(* CoDeSys 2.3.9.47 project: mqtt.pro *)
(* Libraries: Z:\Users\oedemis\Downloads\WagoLibModbus_IP_01.lib 11.2.16 18:05:40, C:\Program Files\WAGO Software\CoDeSys V2.3\Targets\WAGO\Libraries\32_Bit\oscat_basic_333.lib 9.2.16 18:15:54, WagoLibEthernet_01.lib 11.2.16 18:05:44, SysLibSockets.lib 22.5.14 16:16:32, Standard.lib 20.5.14 08:13:26, Iecsfc.lib 16.5.13 14:00:50, SYSLIBCALLBACK.LIB 16.5.13 14:00:50 *)

(* PLC configuration (modules and I/O channels)
K-Bus [K_Bus] node 0, in %IB0 out %QB0 {KbusBusMode = 1; KbusCycleTime = 10000; KbusThreadPriority = 0; KbusSetOutputsToZeroOnApplicationStop = 1}
Modbus variables [PFC200MODBUS] node 1, in %IB0 out %QB0 {PlcStopBehaviour = 1; FiledbusErrorBehaviour = 1; TcpOperation = 1; TcpPort = 502; TcpTimeout = 600; UdpOperation = 1; UdpPort = 502; RtuOperation = 0; NodeId = 1; ResponseTimeout = 5000; Interface = 0; Baud = 115200; StopBits = 1; Parity = 1; FlowCtrl = 0; PhysInterface = 0}
unused [PFC200CANOPEN_UNUSED] node 2, in %IB6000 out %QB6000
Modbus-Master [MB_MASTER] node 3, in %IB0 out %QB0
*)

(* Task configuration *)
TASK Schedule (PRIORITY := 31, INTERVAL := T#100ms);
	PLC_PRG();
END_TASK

(* Global variable list: Globale_Variablen *)
VAR_GLOBAL
	xxSubscribe: BOOL := TRUE;
	xxPublish : BOOL     := TRUE;
	SubPubState : INT;
END_VAR

(* Data type *)
TYPE Buffer :
STRUCT
	data : ARRAY [0..MAX_RECEIVE_TCP_CLIENT] OF BYTE;
	iPos : DWORD := 0;
END_STRUCT
END_TYPE

(* Data type *)
TYPE ConnectFlags :
STRUCT
	xUsername     : BOOL;
	xPassword     : BOOL;
	xWillRetain   : BOOL;
	xWillQoS1     : BOOL;
    xWillQoS2     : BOOL;
	xWillFlag     : BOOL;
	xCleanSession : BOOL;
END_STRUCT
END_TYPE

(* Data type *)
TYPE FixedHeader :
STRUCT
	bMessageType : BYTE := 16#00;
	xDUP_FLAG    : BOOL := FALSE;
	xQos         : BYTE := 16#00; (*0,1,2*)
	xRetain      : BOOL := FALSE;
END_STRUCT
END_TYPE

(* Data type *)
TYPE FixedHeaderSub :
STRUCT
	bMessageType : BYTE := 8;
	xReserved         : BYTE := 2;
END_STRUCT
END_TYPE

(* Data type *)
TYPE Payload :
STRUCT
	data : ARRAY [0..30] OF BYTE;
	iPos : DWORD := 0;
END_STRUCT
END_TYPE

(* POU PLC_PRG, ST *)
PROGRAM PLC_PRG
VAR
	mqttClient: MQTT_Client;
	xPublish: BOOL;
	xSubscribe: BOOL;

	mqttClientFeedIN : MQTT_Client;
	xPublishFeedIN : BOOL;
	xSubscribeFeedIN : BOOL;

	mqttClient2 : MQTT_Client;
	xPublish2 : BOOL;
	xSubscribe2 : BOOL;

	(*Modbus Communication*)
	KOMMU_E: ETHERNET_MODBUSMASTER_TCP;
	Receive_Data: ARRAY [0..5] OF WORD;
	Transmit_Data: ARRAY [0..3] OF WORD;
	TON1:TON;
	diActivePowerSetpoint:DINT;
	xSend:BOOL := TRUE;

	(*test variables*)
	dummy:DATE_AND_TIME;
	str:STRING;
	x:DATE_AND_TIME;
	y:DATE_AND_TIME;
	z:INT;
END_VAR
mqttClient(
xPublish := xxPublish, (* I/O variable to publish to a TOPIC *)
xSubscribe := xxSubscribe,  (* NOT SUPPORTED, but must be here for I/O *)
sIP:='10.210.10.60', (* IP of the MQTT Broker *)
wPortNumber:=1883,  (* PORT of the MQTT Broker *)
(* AUTH: When no authentication is needed, leave the following fields Blank *)
sUsername:='',  (* Username to connect with the MQTT Broker *)
sPassword:='' (* password to connect with the MQTT Broker *)
);

(*mqttClient.sTopic := 'residual/2015-02-13 09:00:00';*)
mqttClient.sTopic := 'residual/+';
mqttClient.sQoS := 16#00;
mqttClient.pTopic := 'pub';
mqttClient.pQoS := 16#00;
mqttClient.pRetained := FALSE;
mqttClient.pPayload := 'wow';


dummy := STRING_TO_DT('DT#2015-02-13-09:00:15');
str:=DT_TO_STRING(DT#1998-02-13-14:20);
x:= SET_DT(
	year := 2015,
	month := 02,
	day := 13  ,
	HOUR := 09,
	MINUTE := 00,
	SECOND := 00);

y:= SET_DT(
	year := 2015,
	month := 02,
	day := 13  ,
	HOUR := 09,
	MINUTE := 00,
	SECOND := 15);

z := DT_TO_INT(y)-DT_TO_INT(x);

(*z:=SECOND_OF_DT(x) - SECOND_OF_DT(y);*)



(*mqttClientFeedIN(
xPublish := xPublishFeedIN, (* I/O variable to publish to a TOPIC *)
xSubscribe := xPublishFeedIN,  (* NOT SUPPORTED, but must be here for I/O *)
sIP:='10.210.10.60', (* IP of the MQTT Broker *)
wPortNumber:=1883,  (* PORT of the MQTT Broker *)
(* AUTH: When no authentication is needed, leave the following fields Blank *)
sUsername:='',  (* Username to connect with the MQTT Broker *)
sPassword:='' (* password to connect with the MQTT Broker *)
);
mqttClientFeedIN.sTopic := 'feedInLimit';
mqttClientFeedIN.sQoS := 16#00;*)

(*Modbus Communication*)

(*diActivePowerSetpoint := mqttClient.activePowerVal;      REAL zu DINT*)

(*KOMMU_E(
  xCONNECT       := TRUE,
  strIP_ADDRESS  := '10.210.10.69',
  wPORT          := 502,
  bUNIT_ID       := 3,
  bFUNCTION_CODE := 16#10,
  wWRITE_ADDRESS := 40149,
  wWRITE_QUANTITY:= 2,
  ptSEND_DATA    := ADR(diActivePowerSetpoint),
  xSEND          := xSend
);*)
END_PROGRAM

(* POU MQTT_Client, ST *)
FUNCTION_BLOCK MQTT_Client
VAR CONSTANT
	VERSION 	: BYTE := 16#03;
	Reserved   	: BYTE := 0;
	CONNECT     : BYTE := 1;
	CONNACK     : BYTE := 2;
	PUBLISH     : BYTE := 3;
	PUBACK      : BYTE := 4;
	PUBREC      : BYTE := 5;
	PUBREL      : BYTE := 6;
	PUBCOMP     : BYTE := 7;
	SUBSCRIBE   : BYTE := 8;
	SUBACK      : BYTE := 9;
	UNSUBSCRIBE : BYTE := 10;
	UNSUBACK    : BYTE := 11;
	PINGREQ     : BYTE := 12;
	PINGRESP    : BYTE := 13;
	DISCONNECT  : BYTE := 14;
	Reserved2   : BYTE := 15;

	CONNECTED   : INT := 30;
	NOT_CONNECTED: INT := 40;
	TIMEOUT : INT := 50;
	WAIT_RESPONSE : INT := 60;

	CONNECTION_TIMEOUT : TIME := t#10s;

	SUBSCRIBED : INT := 70;
	PUBLISHED : INT := 80;
	WAIT_RESPONSE_PUBLISH : INT := 90;
END_VAR

VAR
	fixedHeaderSub : BYTE;
	sendBuffer : Buffer;
	receiveBuffer : Buffer;
	fixedHeader: FixedHeader;
	variableHeader: Buffer;
	payLoad:  Buffer;
	connectFlags: ConnectFlags;
	tcpClient: TCP_Client;
	xTcpConnected: BOOL := FALSE;
	xStartSend: BOOL := FALSE;
	diReceiveCount: DINT;
	connectionTimer: TON;
	xTimeOut: BOOL;
	incomingMessageType: BYTE;
	eState: INT;
	xStartTimer: BOOL;

	a : Buffer;
	b : Buffer;
	i :  DINT := 0;
	j:   DINT;
	x:  INT;
	pValue : REAL; (*Received payload*)
	pValues : ARRAY[0..30] OF BYTE; (* must be reduced  30 zu viel !!!!!!!!!!!!!!!!!!!!!!!!!!!!!!!!!!!!!!!!!!!*)
	timestampPayload : ARRAY[0..13] OF BYTE;
	timestampPreviousPayload : ARRAY[0..13] OF BYTE;
	integral : REAL := 0.0;
	timestamp : DATE_AND_TIME;
	timestampPrev :DATE_AND_TIME;
	deltaT : INT;
	pValueSum : REAL;
	(*payload2 : Payload;*)
	tstart : TOD;
	tstop : TOD;
	tt : TOD;
	c : BOOL;
	(*xPublishTimeOut: BOOL;*)
END_VAR

VAR_INPUT
	sTopic: STRING;
	pTopic: STRING;
	pPayload: STRING;
	pRetained : BOOL;
	pQoS : BYTE;
	sQoS : BYTE;
	sIp : STRING;
	wPortNumber : WORD;
	sUsername : STRING;
	sPassword : STRING;
END_VAR

VAR_IN_OUT
	xPublish: BOOL;
	xSubscribe: BOOL;
END_VAR

VAR_OUTPUT
	xConnected : BOOL := FALSE;
	xBusy : BOOL := FALSE;
	activePowerVal : REAL;
END_VAR
(*_ARRAY_INIT(ADR(receiveBuffer), SIZEOF(receiveBuffer), 0);*)

tcpClient.sIPaddress := sIp;
tcpClient.wPortNumber := wPortNumber;

tcpClient.ptSendData := ADR(sendBuffer.data);
tcpClient.diSendCount := sendBuffer.iPos;

tcpClient(xOpenConnection:=TRUE,
xStartSend:=xStartSend,
aReceiveBuffer := receiveBuffer.data,
diReceiveCount := diReceiveCount);

xTcpConnected := tcpClient.xConnected;
xBusy := xStartSend;

IF NOT xTcpConnected THEN
	eState := NOT_CONNECTED;
	xConnected := FALSE;
 	RETURN;
END_IF;

(* INIT *)
payLoad.iPos := 0;
variableHeader.iPos := 0;

connectionTimer(IN:=xStartTimer, PT:=CONNECTION_TIMEOUT-t#2s);
xTimeOut := connectionTimer.Q;

(*publishTimer(IN := xStartPublishTimer, PT := CONNECTION_TIMEOUT-t#5s);
xPublishTimeOut := publishTimer.Q;
(*Calculate redivelery*)
IF xPublishTimeOut THEN
END_IF*)

tstart := SET_TOD(HOUR:= 09, MINUTE := 00, SECOND:= 00);
tstop := SET_TOD(HOUR:= 15, MINUTE := 00, SECOND:= 00);


(* Calculate the current state *)
IF xTimeOut THEN
	eState := TIMEOUT;
ELSIF eState <> CONNECTED AND eState <> TIMEOUT AND eState <> WAIT_RESPONSE THEN
	eState := NOT_CONNECTED;
END_IF

(* Execute current state *)
CASE eState OF

CONNECTED:
	IF diReceiveCount <> 0 THEN
		incomingMessageType := receiveBuffer.data[0];
		IF incomingMessageType = SHL(PINGRESP, 4) THEN
			xStartTimer := TRUE;
		END_IF
		IF incomingMessageType = SHL(PUBLISH, 4)  THEN
			_ARRAY_INIT(ADR(a), SIZEOF(a), 0);
			_ARRAY_INIT(ADR(pValues), SIZEOF(pValues), 0);
			FOR i:=0 TO diReceiveCount-1 BY 1 DO
				a.data[i] := receiveBuffer.data[i];
			END_FOR
			(*extract payload*)
			i := 0;
			FOR j := 4+a.data[3] TO a.data[1]+1 BY 1 DO
				pValues[i] := a.data[j];
                        		i := i +1 ;
			END_FOR
			(*_PAYLOAD_PUSH(ADR(payload2), pValues);*)
			pValue := CONVERT_TO_REAL(pValues);
			activePowerVal := pValue;
			(*extract timestamp*)
			(*dd := ARRAY_SUM(ADR(timestampPayload), SIZEOF(timestampPayload));*)
			IF timestampPayload[0] <> 0 THEN
				FOR i:=0 TO 13 BY 1 DO
					timestampPreviousPayload[i] := timestampPayload[i];
				END_FOR
				timestampPrev :=  timestamp; (*EXTRACT_TIMESTAMP_FROM_PAYLOAD(timestampPreviousPayload); (*timestamp*)*)
				deltaT := 0;
			END_IF
			i := 0;
			FOR x := 13 TO 31 BY 1 DO
				IF x <> 17 AND x <> 20 AND x <> 23 AND x <> 26 AND x <> 29 THEN
						timestampPayload[i] := a.data[x];
					i := i + 1;
				END_IF
			END_FOR
			timestamp := EXTRACT_TIMESTAMP_FROM_PAYLOAD(timestampPayload);
			(*deltaT := DT_TO_INT(timestamp) - DT_TO_INT(timestampPrev);*)
			(*calculate feed_in_limit*)
			tt := DT_TO_TOD(timestamp);
			(*IF HOUR_OF_DT(timestamp) >= 9 AND  HOUR_OF_DT(timestamp) <= 15 THEN (*alternativ period function of oscat*)*)
			IF TIMECHECK(TD := tt, START := tstart , STOP := tstop) THEN
				(*delta calculation put here*)
				IF YEAR_OF_DATE(DT_TO_DATE(timestampPrev)) <> 1970 THEN deltaT := DT_TO_INT(timestamp) - DT_TO_INT(timestampPrev); END_IF (*Ausreißer in sec umwandeln??? IF deltaT > 900 (15 min) THEN deltaT := 0; END_IF*)
				pValueSum := pValue * deltaT;
				integral := integral + pValueSum;
			END_IF
			(*integral := integral + P_FEED_IN_LIMIT(pValue);*)
		END_IF

		IF incomingMessageType = SHL(PUBACK, 4)  THEN
			_ARRAY_INIT(ADR(b), SIZEOF(b), 0);
			FOR i:=0 TO diReceiveCount-1 BY 1 DO
				b.data[i] := receiveBuffer.data[i];
			END_FOR
		END_IF

		diReceiveCount := 0;
	END_IF

	c := xxPublish AND xxSubscribe;
	IF   c   THEN
		SubPubState := SUBSCRIBED;
	ELSE
		SubPubState := PUBLISHED;
	END_IF;

	CASE SubPubState OF
			SUBSCRIBED:
				IF xxSubscribe THEN
					_BUFFER_CLEAR(ADR(sendBuffer), SIZEOF(sendBuffer));

					fixedHeaderSub :=  BYTE_OF_BIT(FALSE, TRUE, FALSE, FALSE, FALSE, FALSE, FALSE, TRUE); (*FIXED_HEADER*)
					(*fixedHeaderSub.bMessageType := SUBSCRIBE;*)

					_BUFFER_PUSH(ADR(variableHeader), 16#00);(* Message ID *)
					_BUFFER_PUSH(ADR(variableHeader), 16#00);

					_BUFFER_PUSH_STRING(ADR(payLoad), sTopic, TRUE);
					_BUFFER_PUSH(ADR(payLoad), sQoS); (*QoS 0 16#00*);

					sendBuffer.iPos := 0;
					CREATE_MESSAGE_SUB(ADR(sendBuffer), fixedHeaderSub, variableHeader, payLoad);

					xxSubscribe := FALSE;
					(**xxSubscribe := TRUE;**)
					xStartSend := TRUE;
					SubPubState := PUBLISHED;
				END_IF

			 PUBLISHED:
				IF xxPublish THEN
					fixedHeader.bMessageType := PUBLISH;
					fixedHeader.xDUP_FLAG := FALSE;
					(*fixedHeader.xQos := 16#00; (* only QoS 0 supported *)*)
					fixedHeader.xQoS := pQoS;
					fixedHeader.xRetain := pRetained;

					_BUFFER_PUSH_STRING(ADR(variableHeader), pTopic, TRUE); (* Topic *)
					IF fixedHeader.xQos > 16#00 THEN
						_BUFFER_PUSH(ADR(variableHeader), 16#00);(* Message ID *)
						_BUFFER_PUSH(ADR(variableHeader), 16#00);
					END_IF

					_BUFFER_PUSH_STRING(ADR(payLoad), pPayload, FALSE);
					(*_BUFFER_PUSH(ADR(payLoad), sQoS); (*QoS 0 16#00*);*)

					sendBuffer.iPos := 0;
					CREATE_MESSAGE(ADR(sendBuffer), fixedHeader, variableHeader, payLoad);

					xxPublish := TRUE;
					xxSubscribe := TRUE;
					SubPubState := SUBSCRIBED;
					xStartSend := TRUE;
				END_IF
	END_CASE

NOT_CONNECTED:
	sendBuffer.iPos := 0;
	xStartTimer := FALSE;
	fixedHeader.bMessageType := CONNECT;

	_BUFFER_PUSH_STRING(ADR(variableHeader),'MQIsdp', TRUE); (* Protocol Name*)
	_BUFFER_PUSH(ADR(variableHeader), 3); (* Version Number*)

	connectFlags.xCleanSession := TRUE;
	connectFlags.xWillFlag     := FALSE;
	connectFlags.xWillQoS1     := FALSE;
	connectFlags.xWillQoS2     := FALSE;
	connectFlags.xWillRetain   := FALSE;
	IF LEN(sUsername) > 0 THEN
		connectFlags.xUsername := TRUE;
	ELSE
		connectFlags.xUsername := FALSE;
	END_IF
	IF LEN(sPassword) > 0 THEN
		connectFlags.xPassword := TRUE;
	ELSE
		connectFlags.xPassword := FALSE;
	END_IF

	_BUFFER_PUSH(ADR(variableHeader), BYTE_OF_BIT(FALSE,
															connectFlags.xCleanSession,
															connectFlags.xWillFlag,
															connectFlags.xWillQoS1,
															connectFlags.xWillQoS2,
															connectFlags.xWillRetain,
															connectFlags.xPassword,
															connectFlags.xUsername));

	_BUFFER_PUSH(ADR(variableHeader), 16#00);
	_BUFFER_PUSH(ADR(variableHeader), 16#0A); (* Keep Alive: 10s *)

	_BUFFER_PUSH_STRING(ADR(payload), 'PLC', TRUE); (* Client Identfier *)

	IF connectFlags.xUsername THEN
		_BUFFER_PUSH_STRING(ADR(payload), sUsername, TRUE); (* Username *)
	END_IF

	IF connectFlags.xPassword THEN
		_BUFFER_PUSH_STRING(ADR(payload), sPassword, TRUE); (* Password *)
	END_IF

	CREATE_MESSAGE(ADR(sendBuffer), fixedHeader, variableHeader, payLoad);

	eState := WAIT_RESPONSE;
	xStartSend := TRUE;

TIMEOUT:
	sendBuffer.iPos := 0;
	xStartTimer := FALSE;
	fixedHeader.bMessageType := PINGREQ;
	CREATE_MESSAGE(ADR(sendBuffer), fixedHeader, variableHeader, payLoad);

	eState := CONNECTED;
	xStartSend := TRUE;

WAIT_RESPONSE:
	incomingMessageType := receiveBuffer.data[0];
	IF incomingMessageType = SHL(CONNACK, 4) THEN
		(* TODO: Check return code *)
		xConnected := TRUE;
		xStartTimer := TRUE;
		eState := CONNECTED;
		diReceiveCount := 0;
	END_IF
END_CASE
END_FUNCTION_BLOCK

(* POU CONVERT_TO_REAL, ST *)
FUNCTION CONVERT_TO_REAL : REAL
VAR_INPUT
	arTestArray: ARRAY[0..30] OF BYTE;
END_VAR
VAR
	pTestString: POINTER TO STRING;
	rRealValue: REAL;
END_VAR
pTestString:= ADR(arTestArray);

rRealValue:= STRING_TO_REAL(pTestString^);

CONVERT_TO_REAL := rRealValue;
END_FUNCTION

(* POU EXTRACT_TIMESTAMP_FROM_PAYLOAD, ST *)
FUNCTION EXTRACT_TIMESTAMP_FROM_PAYLOAD : DATE_AND_TIME
VAR_INPUT
	data: ARRAY[0..13] OF BYTE;
END_VAR
VAR
	pTestString: POINTER TO STRING;
	pTestStringA: ARRAY[0..5] OF POINTER TO STRING;
	timestamp: DATE_AND_TIME;
	i: INT := 0;
	j : INT := 0;
	yeara : ARRAY[0..4] OF BYTE;
	montha : ARRAY[0..2] OF BYTE;
	daya : ARRAY[0..2] OF BYTE;
	houra : ARRAY[0..2] OF BYTE;
	minutea : ARRAY[0..2] OF BYTE;
	seconda : ARRAY[0..2] OF BYTE;

	year1: INT;
	month1: INT;
	day1: INT;
	hour1: INT;
	minute1:INT;
	second1:INT;

	rRealValue: BOOL;
END_VAR
FOR i := 0 TO 13 BY 1 DO
	IF i <= 3				 		THEN yeara[i] := data[i];
	ELSIF  i > 3 AND i <= 5 			THEN IF j > 1 THEN j := 0;  END_IF; 		montha[j] := data[i];  	 j:=j+1;
	ELSIF  i > 5 AND i <= 7 			THEN IF j > 1 THEN j := 0;  END_IF;  	daya[j] := data[i]; 	 j:=j+1;
	ELSIF  i >= 8 AND i <= 9 			THEN IF j > 1 THEN j := 0;  END_IF; 		houra[j] := data[i];   	 j:=j+1;
	ELSIF  i > 9 AND i <= 11 			THEN IF j > 1 THEN j := 0;  END_IF; 		minutea[j] := data[i];   j:=j+1;
	ELSIF  i > 11 AND i <= 13 		THEN IF j > 1 THEN j := 0;   END_IF;  	seconda[j] := data[i];  j:=j+1;
	END_IF;
END_FOR

(*pTestString:= ADR(yeara);
iValue:= STRING_TO_INT(pTestString^);
EXTRACT_TIMESTAMP_FROM_PAYLOAD := iValue;*)

pTestStringA[0] := ADR(yeara);
pTestStringA[1] := ADR(montha);
pTestStringA[2] := ADR(daya);
pTestStringA[3] := ADR(houra);
pTestStringA[4] := ADR(minutea);
pTestStringA[5] := ADR(seconda);

(*pTestString	 :=      ADR(yeara);
year1		 :=  	STRING_TO_INT(pTestString^);
EXTRACT_TIMESTAMP_FROM_PAYLOAD := year1;*)

year1:=  		STRING_TO_INT(pTestStringA[0]^);
month1 :=  	STRING_TO_INT(pTestStringA[1]^);
day1 := 		STRING_TO_INT(pTestStringA[2]^);
hour1 := 		STRING_TO_INT(pTestStringA[3]^);
minute1 := 	STRING_TO_INT(pTestStringA[4]^);
second1 :=  	STRING_TO_INT(pTestStringA[5]^);


EXTRACT_TIMESTAMP_FROM_PAYLOAD := SET_DT(
	year := year1,
	month := month1,
	day := day1  ,
	HOUR := hour1,
	MINUTE := minute1,
	SECOND := second1);
END_FUNCTION

(* POU _BUFFER_PUSH, ST *)
FUNCTION _BUFFER_PUSH : BOOL
VAR_INPUT
	PT  : POINTER TO Buffer;
	IN  : BYTE;
END_VAR

VAR
END_VAR
(* pushed data to a buffer array *)
PT^.data[PT^.iPos] := IN;

PT^.iPos := PT^.iPos + 1;

_BUFFER_PUSH := TRUE;
END_FUNCTION

(* POU _BUFFER_PUSH_STRING, ST *)
FUNCTION _BUFFER_PUSH_STRING : BOOL
VAR_INPUT
	PT : POINTER TO Buffer;
	IN : STRING;
	INCLUDE_LENGTH : BOOL := FALSE;
END_VAR
VAR
	sPT : POINTER TO BYTE;
	iLen : DWORD;
	i : DWORD;
	nxtPtr: POINTER TO BYTE;
END_VAR
iLen := LEN(IN);
sPT := ADR(IN);

IF INCLUDE_LENGTH THEN
	_BUFFER_PUSH(PT, BYTE_OF_DWORD(iLen,1));
	_BUFFER_PUSH(PT, BYTE_OF_DWORD(iLen,0));
END_IF

FOR i:=0 TO iLen-1 BY 1 DO
	nxtPtr := sPT + i * SIZEOF(sPT^);
	_BUFFER_PUSH(PT, nxtPtr^);
END_FOR
END_FUNCTION

(* POU CREATE_MESSAGE_SUB, ST *)
FUNCTION CREATE_MESSAGE_SUB : BOOL
VAR_INPUT
	PT          			:POINTER TO Buffer;
	fixedHeader      	: BYTE;
	variableHeader  	:Buffer;
	payLoad         		:Buffer;
END_VAR
VAR
	bTemp  			:BYTE;
	remainingLength	:DWORD;
END_VAR
(* FIXED HEADER *)
(* BYTE 1 *)
(*bTemp := bTemp OR SHL(fixedHeader, 4);*)
(*bTemp := bTemp OR fixedHeader;*)
bTemp := fixedHeader;

_BUFFER_PUSH(PT, bTemp);

(* BYTE 2 *)
remainingLength := variableHeader.iPos + payLoad.iPos;

ENCODE_REMAINING_LENGTH(PT, remainingLength);
(*_BUFFER_PUSH(PT, remainingLength);*)

(* VARIABLE HEADER *)
_BUFFER_CONCAT(PT, ADR(variableHeader));

(* PAYLOAD *)
_BUFFER_CONCAT(PT, ADR(payLoad));
END_FUNCTION

(* POU ENCODE_REMAINING_LENGTH, ST *)
FUNCTION ENCODE_REMAINING_LENGTH : BOOL
VAR_INPUT
	PT : POINTER TO Buffer;
	LENGTH : DWORD;
END_VAR
VAR
	wPt : POINTER TO DWORD; (*4 bytes*)
	digit: DWORD;
	i: UINT;
END_VAR
wPt := ADR(LENGTH);

IF LENGTH = 0 THEN
	_BUFFER_PUSH(PT, 16#00);
	RETURN;
END_IF

WHILE LENGTH > 0 DO
	digit := LENGTH MOD 128;
	LENGTH := LENGTH / 128;
	
	IF LENGTH > 0 THEN
		digit := digit OR 16#80;
	END_IF
	_BUFFER_PUSH(PT, BYTE_OF_DWORD(digit,0));
END_WHILE
END_FUNCTION

(* POU _BUFFER_CONCAT, ST *)
FUNCTION _BUFFER_CONCAT : BOOL
VAR_INPUT
	PT  : POINTER TO Buffer;
	PTContact  : POINTER TO Buffer;
END_VAR
VAR
	i: INT;
END_VAR
FOR i:=0 TO DWORD_TO_INT(PTContact^.iPos) -1 BY 1 DO
	_BUFFER_PUSH(PT, PTContact^.data[i]);
END_FOR
END_FUNCTION

(* POU CREATE_MESSAGE, ST *)
FUNCTION CREATE_MESSAGE : BOOL
VAR_INPUT
	PT          : POINTER TO Buffer;
	fixedHeader     : FixedHeader;
	variableHeader  : Buffer;
	payLoad         : Buffer;
END_VAR
VAR
	bTemp  : BYTE;
	remainingLength: DWORD;
END_VAR
(* FIXED HEADER *)
(* BYTE 1 *)
bTemp := bTemp OR SHL(fixedHeader.bMessageType, 4) OR SHL(FixedHeader.xQos, 1);

BIT_LOAD_B(bTemp, FixedHeader.xDUP_FLAG, 3);
BIT_LOAD_B(bTemp, FixedHeader.xRetain, 0);

_BUFFER_PUSH(PT, bTemp);

(* BYTE 2 *)
remainingLength := variableHeader.iPos + payLoad.iPos;

ENCODE_REMAINING_LENGTH(PT, remainingLength);
(*_BUFFER_PUSH(PT, remainingLength);*)

(* VARIABLE HEADER *)
_BUFFER_CONCAT(PT, ADR(variableHeader));

(* PAYLOAD *)
_BUFFER_CONCAT(PT, ADR(payLoad));
END_FUNCTION

(* POU _BUFFER_SET, ST *)
FUNCTION _BUFFER_SET : BOOL
VAR_INPUT
	PT  : POINTER TO Buffer;
	IN  : BYTE;
	POS : UINT := 0;
END_VAR
VAR
END_VAR
PT^.data[POS] := IN;

IF PT^.iPos < POS THEN
	PT^.iPos := POS;
END_IF
END_FUNCTION

(* POU _PAYLOAD_PUSH, ST *)
FUNCTION _PAYLOAD_PUSH : BOOL
VAR_INPUT
	PT  : POINTER TO Payload;
	IN  : BYTE;
END_VAR
VAR
END_VAR
(* pushed data to a buffer array *)
PT^.data[PT^.iPos] := IN;

PT^.iPos := PT^.iPos + 1;

_PAYLOAD_PUSH := TRUE;
END_FUNCTION

(* POU P_FEED_IN_LIMIT, ST *)
FUNCTION P_FEED_IN_LIMIT : REAL
VAR_INPUT
	p_Residual_T_Integral: REAL;
	Q_Battery_Full : REAL;
	tStart: INT;
	tStop: INT;
	(*pVals: ARRAY[0..30] OF BYTE;*)
END_VAR
VAR
	i : REAL;
	(*PF : FT_INT2;*)
END_VAR
P_FEED_IN_LIMIT := (p_Residual_T_Integral - Q_Battery_Full) / (tStart - tStop);


(*PF(
	IN:= p_Residual_T ,
	K:= 1.0,
	RUN:= TRUE,
	(*RST:= ,*)
	OUT_MIN:=t_Start,
	OUT_MAX:=t_Stop);

P_FEED_IN_LIMIT := PF.OUT;*)

(*P_FEED_IN_LIMIT := 0.1;*)
END_FUNCTION
